{attribute 'linkalways'}
{attribute 'no_explicit_call' := 'do not call this POU directly'}
FUNCTION_BLOCK ABSTRACT CyclicInstance EXTENDS Instance IMPLEMENTS I_CyclicInstance
VAR
	membership : AutomaticGlobalInstanceMembership(THIS^);
	_cyclicInstanceCallback : CyclicCallback(THIS^);
END_VAR

METHOD ABSTRACT CyclicCall
VAR_INPUT
END_VAR
END_METHOD

PROPERTY PUBLIC CyclicInstanceCallback : I_Callback
GET
CyclicInstanceCallback := _cyclicInstanceCallback;
END_GET
END_PROPERTY

END_FUNCTION_BLOCK

(* stored: Version 1.1.0.1, ProductVersion 3.1.4024.11
   POU CyclicInstance: Id {dc2e84c3-6d56-43a2-a4f0-a82e4ef40050}, SpecialFunc None
   Folder Abstract: Id {25661d79-aab9-4fb7-bdb4-976335c48e7a}
   Method CyclicCall: Id {88412bc0-cc27-4015-9d40-0dabd1437f7c}
   Property CyclicInstanceCallback: Id {2fedc0eb-3da0-43a8-8555-691afde2d4a4}
   Get Get: Id {49d5d242-2da3-436f-b409-782c762f0a38} *)
